FUNCTION_BLOCK TwoConCtlRingHead (* Composite Function Block Type *)
  (* Standard: 61499-2 *)
  (* Version 0.2, 2003-12-05, JHC, Rockwell Automation, Renamed from NEWCOMPFB. *)
  (* Version 0.1, 2002-01-08, JHC, Rockwell Automation, Added DLY FB as example. *)
  (* Version 0.0, 2000-05-27, JHC, Rockwell Automation *)
  (* Compiler header: package fb.rt.cs725; *)
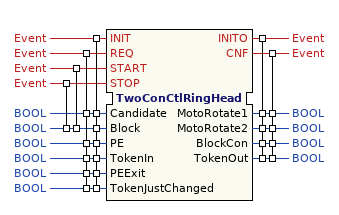
  EVENT_INPUT
    INIT WITH Candidate, Block, PE, TokenIn, PEExit, TokenJustChanged; (* Initialization Request *)
    REQ WITH Candidate, PE, TokenIn, PEExit, TokenJustChanged; (* Normal Execution Request *)
    START WITH Block;
    STOP WITH Block;
  END_EVENT
  EVENT_OUTPUT
    INITO WITH MotoRotate1, MotoRotate2, BlockCon, TokenOut; (* Initialization Confirm *)
    CNF WITH MotoRotate1, MotoRotate2, BlockCon, TokenOut; (* Execution Confirmation *)
  END_EVENT
  VAR_INPUT
    Candidate : BOOL;
    Block : BOOL;
    PE : BOOL;
    TokenIn : BOOL;
    PEExit : BOOL;
    TokenJustChanged : BOOL;
  END_VAR
  VAR_OUTPUT
    MotoRotate1 : BOOL;
    MotoRotate2 : BOOL;
    BlockCon : BOOL;
    TokenOut : BOOL;
  END_VAR
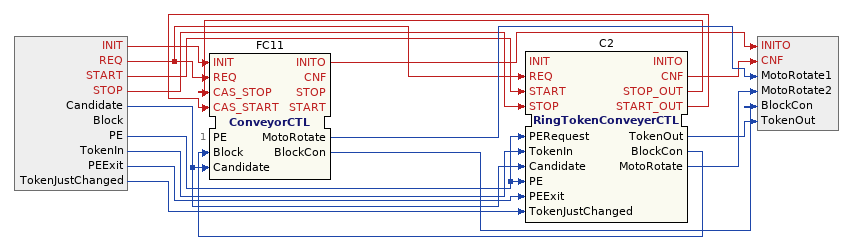
  FBS
    FC11 : ConveyorCTL(PE := 1);
    C2 : RingTokenConveyerCTL;
  END_FBS
  EVENT_CONNECTIONS
    INIT TO FC11.INIT;
    REQ TO FC11.REQ;
    C2.CNF TO CNF;
    C2.STOP_OUT TO FC11.CAS_STOP;
    C2.START_OUT TO FC11.CAS_START;
    START TO C2.START;
    STOP TO C2.STOP;
    REQ TO C2.REQ;
    FC11.INITO TO INITO;
  END_CONNECTIONS
  DATA_CONNECTIONS
    FC11.MotoRotate TO MotoRotate1;
    Candidate TO FC11.Candidate;
    FC11.BlockCon TO BlockCon;
    C2.MotoRotate TO MotoRotate2;
    C2.BlockCon TO FC11.Block;
    PE TO C2.PE;
    Candidate TO C2.Candidate;
    PE TO C2.PERequest;
    TokenIn TO C2.TokenIn;
    C2.TokenOut TO TokenOut;
    PEExit TO C2.PEExit;
    TokenJustChanged TO C2.TokenJustChanged;
  END_CONNECTIONS
END_FUNCTION_BLOCK
